// TIA Portal V17 export
// export: Created 2023-02-14T02:49:44.6195475Z, ExportSetting WithDefaults, DisplayName Totally Integrated Automation Portal, DisplayVersion V17, DisplayName TIA Portal Openness, DisplayVersion V17, DisplayName TIA Portal Teamcenter Gateway, DisplayVersion V17, DisplayName TIA Portal Version Control Interface, DisplayVersion V17, DisplayName SINAMICS Startdrive Advanced, DisplayVersion V17, DisplayName SINAMICS Startdrive G130, G150, S120, S150, SINAMICS MV, S210, DisplayVersion V17, DisplayName SINAMICS Startdrive G110M, G120, G120C, G120D, G120P, G115D, DisplayVersion V17, DisplayName STEP 7 Professional, DisplayVersion V17, DisplayName STEP 7 Safety, DisplayVersion V17, DisplayName WinCC Professional, DisplayVersion V17
FUNCTION_BLOCK "Alarm_Collector_Gen"   // FB33, LAD
{ S7_Optimized_Access := 'TRUE' }
VERSION : 0.1
// stored: AutoNumber true, IsIECCheckEnabled false, IsRetainMemResEnabled false, MemoryReserve 100, SetENOAutomatically false, UDAEnableTagReadback false
   VAR
      Alarm_DRP : DWord;   // Dry Run Protection Alarm
      Alarm_PS : DWord;   // Pressure Switch Alarm
   END_VAR
BEGIN

REGION Network 1: Alarm DRP
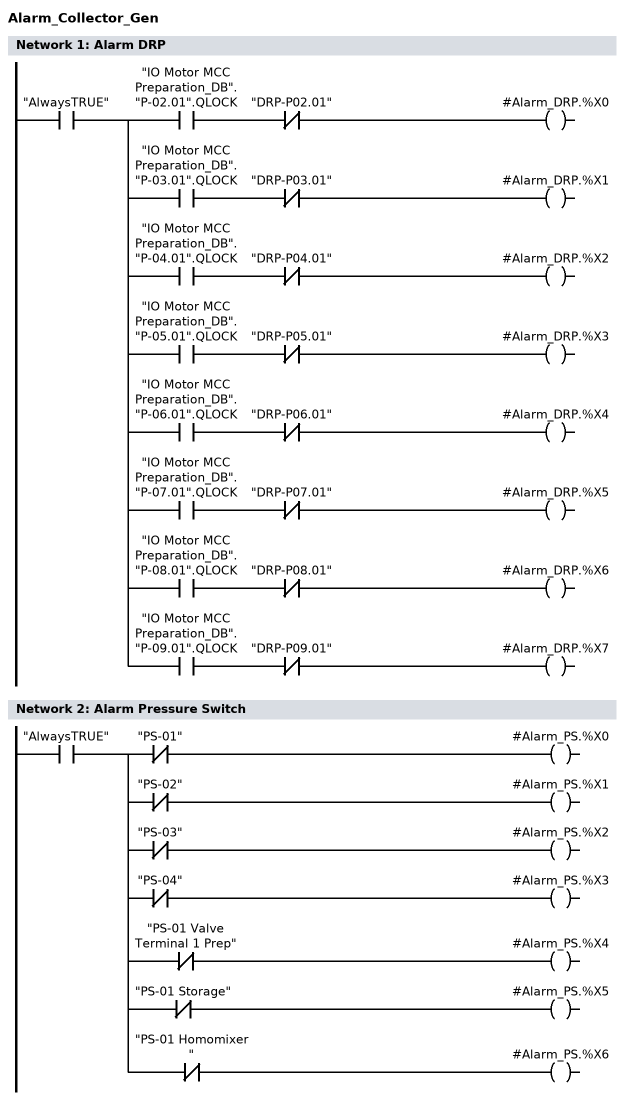
   RUNG wire#powerrail
      Contact( "AlwaysTRUE" )
      wire#w1
      Contact( "IO Motor MCC Preparation_DB"."P-02.01".QLOCK )
      I_Contact( "DRP-P02.01" )
      Coil( #Alarm_DRP.%X0 )
   END_RUNG
   RUNG wire#w1
      Contact( "IO Motor MCC Preparation_DB"."P-03.01".QLOCK )
      I_Contact( "DRP-P03.01" )
      Coil( #Alarm_DRP.%X1 )
   END_RUNG
   RUNG wire#w1
      Contact( "IO Motor MCC Preparation_DB"."P-04.01".QLOCK )
      I_Contact( "DRP-P04.01" )
      Coil( #Alarm_DRP.%X2 )
   END_RUNG
   RUNG wire#w1
      Contact( "IO Motor MCC Preparation_DB"."P-05.01".QLOCK )
      I_Contact( "DRP-P05.01" )
      Coil( #Alarm_DRP.%X3 )
   END_RUNG
   RUNG wire#w1
      Contact( "IO Motor MCC Preparation_DB"."P-06.01".QLOCK )
      I_Contact( "DRP-P06.01" )
      Coil( #Alarm_DRP.%X4 )
   END_RUNG
   RUNG wire#w1
      Contact( "IO Motor MCC Preparation_DB"."P-07.01".QLOCK )
      I_Contact( "DRP-P07.01" )
      Coil( #Alarm_DRP.%X5 )
   END_RUNG
   RUNG wire#w1
      Contact( "IO Motor MCC Preparation_DB"."P-08.01".QLOCK )
      I_Contact( "DRP-P08.01" )
      Coil( #Alarm_DRP.%X6 )
   END_RUNG
   RUNG wire#w1
      Contact( "IO Motor MCC Preparation_DB"."P-09.01".QLOCK )
      I_Contact( "DRP-P09.01" )
      Coil( #Alarm_DRP.%X7 )
   END_RUNG
   // the same network as SCL:
   #Alarm_DRP.%X0 := "AlwaysTRUE" AND "IO Motor MCC Preparation_DB"."P-02.01".QLOCK AND NOT "DRP-P02.01";
   #Alarm_DRP.%X1 := "AlwaysTRUE" AND "IO Motor MCC Preparation_DB"."P-03.01".QLOCK AND NOT "DRP-P03.01";
   #Alarm_DRP.%X2 := "AlwaysTRUE" AND "IO Motor MCC Preparation_DB"."P-04.01".QLOCK AND NOT "DRP-P04.01";
   #Alarm_DRP.%X3 := "AlwaysTRUE" AND "IO Motor MCC Preparation_DB"."P-05.01".QLOCK AND NOT "DRP-P05.01";
   #Alarm_DRP.%X4 := "AlwaysTRUE" AND "IO Motor MCC Preparation_DB"."P-06.01".QLOCK AND NOT "DRP-P06.01";
   #Alarm_DRP.%X5 := "AlwaysTRUE" AND "IO Motor MCC Preparation_DB"."P-07.01".QLOCK AND NOT "DRP-P07.01";
   #Alarm_DRP.%X6 := "AlwaysTRUE" AND "IO Motor MCC Preparation_DB"."P-08.01".QLOCK AND NOT "DRP-P08.01";
   #Alarm_DRP.%X7 := "AlwaysTRUE" AND "IO Motor MCC Preparation_DB"."P-09.01".QLOCK AND NOT "DRP-P09.01";
END_REGION

REGION Network 2: Alarm Pressure Switch
   RUNG wire#powerrail
      Contact( "AlwaysTRUE" )
      wire#w1
      I_Contact( "PS-01" )
      Coil( #Alarm_PS.%X0 )
   END_RUNG
   RUNG wire#w1
      I_Contact( "PS-02" )
      Coil( #Alarm_PS.%X1 )
   END_RUNG
   RUNG wire#w1
      I_Contact( "PS-03" )
      Coil( #Alarm_PS.%X2 )
   END_RUNG
   RUNG wire#w1
      I_Contact( "PS-04" )
      Coil( #Alarm_PS.%X3 )
   END_RUNG
   RUNG wire#w1
      I_Contact( "PS-01 Valve Terminal 1 Prep" )
      Coil( #Alarm_PS.%X4 )
   END_RUNG
   RUNG wire#w1
      I_Contact( "PS-01 Storage" )
      Coil( #Alarm_PS.%X5 )
   END_RUNG
   RUNG wire#w1
      I_Contact( "PS-01 Homomixer" )
      Coil( #Alarm_PS.%X6 )
   END_RUNG
   // the same network as SCL:
   #Alarm_PS.%X0 := "AlwaysTRUE" AND NOT "PS-01";
   #Alarm_PS.%X1 := "AlwaysTRUE" AND NOT "PS-02";
   #Alarm_PS.%X2 := "AlwaysTRUE" AND NOT "PS-03";
   #Alarm_PS.%X3 := "AlwaysTRUE" AND NOT "PS-04";
   #Alarm_PS.%X4 := "AlwaysTRUE" AND NOT "PS-01 Valve Terminal 1 Prep";
   #Alarm_PS.%X5 := "AlwaysTRUE" AND NOT "PS-01 Storage";
   #Alarm_PS.%X6 := "AlwaysTRUE" AND NOT "PS-01 Homomixer";
END_REGION
END_FUNCTION_BLOCK
